{attribute 'qualified_only'}
{attribute 'strict'}
TYPE eHeaderPieces :
(
	Ok 		:= 0,
	Ko 		:= 1,
	Loaded	:= 2,
	Total	:= 3,
	End		:= 4
);
END_TYPE

(* stored: Version 1.1.0.1, ProductVersion 3.1.4024.13
   EnumerationTextList eHeaderPieces: Id {021ec05f-ee7b-4cd6-b387-b07eda5f6a50} *)
